// TIA Portal V17 export
// export: Created 2022-05-25T12:57:42.3003549Z, ExportSetting WithDefaults, DisplayName Totally Integrated Automation Portal, DisplayVersion V17, DisplayName TIA Portal Openness, DisplayVersion V17, DisplayName TIA Portal Version Control Interface, DisplayVersion V17, DisplayName STEP 7 Professional, DisplayVersion V17, DisplayName STEP 7 Safety, DisplayVersion V17, DisplayName WinCC Professional, DisplayVersion V17
VAR_GLOBAL   // PLC tag table "GP25_Yaskawa_Output_Mapping"
   Statusbit_0 AT %I2191.0 : Bool;
   Statusbit_1 AT %I2191.1 : Bool;
   Statusbit_2 AT %I2191.2 : Bool;
   Statusbit_3 AT %I2191.3 : Bool;
   Statusbit_4 AT %I2191.4 : Bool;
   Statusbit_5 AT %I2191.5 : Bool;
   Statusbit_6 AT %I2191.6 : Bool;
   Statusbit_7 AT %I2191.7 : Bool;
   Operating AT %I2192.0 : Bool;
   Servo_on AT %I2192.1 : Bool;
   Top_Of_Master_Job AT %I2192.2 : Bool;
   "Alarm/Error_Occurred" AT %I2192.3 : Bool;
   Reduced_Speed_Input AT %I2192.4 : Bool;
   Remote_Mode_Setting AT %I2192.5 : Bool;
   Play_Mode_Setting AT %I2192.6 : Bool;
   Teach_Mode_Setting AT %I2192.7 : Bool;
   Battery_Alarm AT %I2193.0 : Bool;
   Watchdog_Input AT %I2193.1 : Bool;
   Hold AT %I2193.2 : Bool;
   Shocksensor AT %I2193.3 : Bool;
   Continues_Cycle_Select_Input AT %I2193.4 : Bool;
   "1_Cycle_Selec_Input" AT %I2193.5 : Bool;
   Dialog_Displayed_At_Start AT %I2193.6 : Bool;
   Energy_Saving_Input AT %I2193.7 : Bool;
   Major_Alarm_Occure AT %I2194.0 : Bool;
   Minor_Alarm_Occure AT %I2194.1 : Bool;
   System_Alarm_Occure AT %I2194.2 : Bool;
   User_Alarm_Occure AT %I2194.3 : Bool;
   SAF_Safety_Plug_Input AT %I2194.4 : Bool;
   External_Emergency_Stop AT %I2194.5 : Bool;
   Teach_Box_Emergency_Stop AT %I2194.6 : Bool;
   Extern_Hold AT %I2194.7 : Bool;
   Shock_Detention_On_R1 AT %I2195.0 : Bool;
   In_Cube_1 AT %I2195.1 : Bool;
   In_Cube_2 AT %I2195.2 : Bool;
   In_Cube_3 AT %I2195.3 : Bool;
   In_Cube_4 AT %I2195.4 : Bool;
   In_Cube_5 AT %I2195.5 : Bool;
   In_Cube_6 AT %I2195.6 : Bool;
   In_Cube_7 AT %I2195.7 : Bool;
   In_Cube_8 AT %I2196.0 : Bool;
END_VAR
